// TIA Portal V17 export
// export: Created 2026-04-13T11:12:42.2859329Z, ExportSetting WithDefaults, DisplayName Totally Integrated Automation Portal, DisplayVersion V17 Update 4, DisplayName TIA Portal Openness, DisplayVersion V17 Update 4, DisplayName TIA Portal Version Control Interface, DisplayVersion V17, DisplayName SINAMICS Startdrive Advanced, DisplayVersion V17, DisplayName SINAMICS Startdrive G130, G150, S120, S150, SINAMICS MV, S210, DisplayVersion V17, DisplayName SINAMICS Startdrive G110M, G120, G120C, G120D, G120P, G115D, DisplayVersion V17, DisplayName STEP 7 Professional, DisplayVersion V17 Update 4, DisplayName STEP 7 Safety, DisplayVersion V17, DisplayName WinCC Professional, DisplayVersion V17 Update 4
FUNCTION_BLOCK "5-定时器"   // FB72, SCL
{ S7_Optimized_Access := 'TRUE' }
VERSION : 0.1
// stored: AutoNumber true, IsIECCheckEnabled false, IsRetainMemResEnabled false, MemoryReserve 100, SetENOAutomatically false, UDAEnableTagReadback false
   VAR_INPUT
      计时开始 : Bool;
      定时器设置时间 : Time;
   END_VAR
   VAR_OUTPUT
      剩余时间分 : Int;
      剩余时间秒 : Int;
      计时到达 : Bool;
   END_VAR
   VAR
      定时器当前时间 : Time;
      "TIMER" : TON_TIME;
   END_VAR
   VAR_TEMP
      TEMP剩余时间 : Time;
   END_VAR
BEGIN
   #TIMER(IN:=#计时开始,
          PT:=#定时器设置时间,
          Q=>#计时到达,
          ET=>#定时器当前时间);



   //计时未开始，剩余时间为0
   IF NOT #计时开始 THEN
       #剩余时间分 := 0;
       #剩余时间秒 := 0;
   END_IF;

   IF #定时器当前时间 > t#0ms THEN
       #TEMP剩余时间 := (#定时器设置时间 / 1000)-(#定时器当前时间/1000);
       #剩余时间分 := TIME_TO_INT(#TEMP剩余时间)/60;
       #剩余时间秒 := TIME_TO_INT(#TEMP剩余时间) MOD 60;
   END_IF;
END_FUNCTION_BLOCK
